TYPE STriggeredOutput :
STRUCT
	ChangeTrigger: USINT;
END_STRUCT
END_TYPE

(* stored: Version 1.1.0.1, ProductVersion 3.1.4024.9
   DUT STriggeredOutput: Id {1728715d-7add-4733-b647-77ca6f61d531} *)
